// TIA Portal V16 export
// export: Created 2021-09-15T08:32:33.3605739Z, ExportSetting WithDefaults, DisplayName Totally Integrated Automation Portal, DisplayVersion V16 Update 4, DisplayName TIA Portal Version Control Interface, DisplayVersion V16 Update 2, DisplayName TIA Portal Openness, DisplayVersion V16 Update 4, DisplayName SINAMICS Startdrive Advanced, DisplayVersion V16 Update 5, DisplayName SINAMICS DCC, DisplayVersion V16, DisplayName SINAMICS Startdrive G130, G150, S120, S150, SINAMICS MV, S210, DisplayVersion V16 Update 5, DisplayName SINAMICS Startdrive G110M, G120, G120C, G120D, G120P, G115D, DisplayVersion V16 Update 5, DisplayName STEP 7 Professional, DisplayVersion V16 Update 4, DisplayName STEP 7 Safety, DisplayVersion V16, DisplayName Simocode ES, DisplayVersion V16 Upd2, DisplayName WinCC Advanced / Unified PC, DisplayVersion V16 Update 4
FUNCTION "Main_CyclicApp" : Void   // FC1, FBD
TITLE = Main_CyclicApp
{ S7_Optimized_Access := 'TRUE' }
AUTHOR : A.Cehajic
VERSION : 0.1
// stored: AutoNumber false, IsIECCheckEnabled false, SetENOAutomatically false, UDAEnableTagReadback false
BEGIN

REGION Network 1
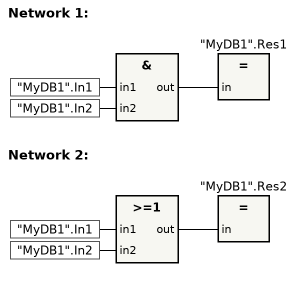
   "MyDB1".Res1 := "MyDB1".In1 AND "MyDB1".In2;
END_REGION

REGION Network 2
   "MyDB1".Res2 := "MyDB1".In1 OR "MyDB1".In2;
END_REGION
END_FUNCTION
